# B&R Automation Studio project SysReset
Automation Studio 4.9

## Configuration TestSetup

CPU X20CP1585, AutomationRuntime C4.90, Build 4.1.2, Vc V4.72.0

### Task classes (Cpu.sw)
```
Cyclic#4:
  DevLinker <- DevLinker.prg
  SysRst <- SysRst.prg
Cyclic#7:
  HelloFile <- HelloFile.prg
Binaries: FWRules, TCData, udbdef, asfw, User, iomap, sysconf, arconfig, ashwd, Role, ashwac
Libraries: sys_lib, runtime, standard, AsSem, FileIO, AsIODiag, asieccon, astime
```

### Hardware
```
X20BM11 : X20BM11 v1.0.0.1  [X2X1 -> X20CP1585.IF6]
X20CP1585 : X20CP1585 v1.8.1.0
  Connector IF2:
    ActivateDevice = 1
    HostName = sysreset
  ConfigurationID = SysReset_Config1
  Simulation = 1
  EthernetHostName = sysreset
  ActivateDns = 1
  GetDnsFromDhcp = 2
X20DI9371 : X20DI9371 v1.1.0.0  [SS1 -> X20TB12.SS; SL -> X20BM11.SL1]
X20TB12 : X20TB12 v1.0.0.0
```

### IoMap.iom - X20CP1585/IoMap.iom
```iecst
VAR_CONFIG
	::SysRst:diVdc24Ok AT %IX."X20DI9371".DigitalInput01;
END_VAR
```

### PvMap.vvm - X20CP1585/PvMap.vvm
```iecst
VAR_CONFIG
	::SysRst:oSemIdent AT %Q.::HelloFile:iSemIdent; (*Insert your comment here...*)
	::SysRst:oFileSystemLocked AT %Q.::HelloFile:iFileSystemLocked; (*Insert your comment here...*)
END_VAR
```

## Logical view

Binary libraries used (declarations not repeated): operator, runtime, astime, AsIecCon, sys_lib, standard, AsSem, FileIO, AsIODiag

### Global.var - Global variables
```iecst
VAR CONSTANT
	FILE_DEVICE_LOCAL : STRING[80] := 'LOCAL';
END_VAR
```


### Program Logical/DevLinker (IEC) - Creates file devices

#### Variables.var
```iecst
VAR
	fbDevLink : DevLink; (*links file device*)
	fbDevUnlink : DevUnlink; (*unlinks file device*)
	fbDirCreate : DirCreate; (*creates directory*)
END_VAR
VAR CONSTANT
	FILE_DEVICE_TEMP : STRING[80] := '__TEMP__'; (*name of temporary file device*)
END_VAR
```

#### Main.st
```iecst
(*********************************************************************************
 * Copyright: B&R Industrial Automation GmbH
 * Author:    knausenbergl
 * Created:   April 12, 2021/1:55 PM

Link a file device on the CF user partition (ArEmb) or in the windows temp folder (ArSim), respectively.
Required for file handling.
 *********************************************************************************)

PROGRAM _INIT

	(* for ArSim, create folder structure under "C:/Temp" *)
	IF DiagCpuIsARsim() OR DiagCpuIsSimulated() THEN
		(* link file device in windows temp folder. this file device is only needed for creating subfolders. *)
		fbDevLink.enable := TRUE;
		fbDevLink.pDevice := ADR(FILE_DEVICE_TEMP);
		fbDevLink.pParam := ADR('/DEVICE=C:/Temp/');
		fbDevLink();

		(* create directory "SysReset" in windows temp folder *)
		fbDirCreate.enable := TRUE;
		fbDirCreate.pDevice := ADR(FILE_DEVICE_TEMP);
		fbDirCreate.pName := ADR('SysReset');
		fbDirCreate();

		(* unlink temporary file device, it is no longer needed *)
		fbDevUnlink.enable := TRUE;
		fbDevUnlink.handle := fbDevLink.handle;
		fbDevUnlink();
	END_IF

	(* link FILE_DEVICE_LOCAL, which is used for data storage by other tasks *)
	fbDevLink.enable := TRUE;
	fbDevLink.pDevice := ADR(FILE_DEVICE_LOCAL);
	IF DiagCpuIsARsim() OR DiagCpuIsSimulated() THEN
		fbDevLink.pParam := ADR('/DEVICE=C:/Temp/SysReset');
	ELSE
		fbDevLink.pParam := ADR('/DEVICE=F:/');
	END_IF
	fbDevLink();

END_PROGRAM

PROGRAM _CYCLIC
	(* Insert code here *)

END_PROGRAM

PROGRAM _EXIT

	fbDevUnlink.enable := TRUE;
	fbDevUnlink.handle := fbDevLink.handle;
	fbDevUnlink();

END_PROGRAM
```

### Program Logical/SysRst (IEC) - Controlled PLC shutdown

#### Main.st - Init, cyclic, exit code
```iecst
(*********************************************************************************
 * Copyright: B&R Industrial Automation GmbH
 * Author:    knausenbergl
 * Created:   January 18, 2021/11:20 AM

This task initiates a controlled shutdown of the PLC if either of the following conditions applies:
1. Drop in 24VDC supply, running on buffered 24VDC supply. (Only applies if buffered 24VDC is used.)
2. Shutdown command triggered, e.g. by visualization.

This task ensures file consistency in the case of a shutdown. This is done via the use of
semaphores. Any task accessing the file system must acquire a semaphore. The shutdown only
starts if the semaphore is no longer in use.
 *********************************************************************************)

PROGRAM _INIT

	(* create semaphore for detecting usage of file system *)
	fbSemCreate.enable		:= TRUE;
	fbSemCreate.maxCount	:= SEM_MAX_COUNT;
	fbSemCreate.initCount	:= fbSemCreate.maxCount;
	fbSemCreate();
	oSemIdent	:= fbSemCreate.ident;

	TOF_Vdc24Ok.PT	:= VDC24_OK_OFF_DELAY;

END_PROGRAM

PROGRAM _CYCLIC

	TOF_Vdc24Ok(IN := diVdc24Ok);			//off-delay for "24VDC OK" signal to filter short drops in 24VDC power supply
	F_TRIG_Vdc24Ok(CLK := TOF_Vdc24Ok.Q);	//falling edge of filtered "24VDC OK" signal

	(* check if file system is busy *)
	fbSemGetInfo.enable	:= TRUE;
	fbSemGetInfo.ident	:= fbSemCreate.ident;
	fbSemGetInfo();
	FileSystemBusy	:= (fbSemGetInfo.maxCount <> fbSemGetInfo.curCount);

	(* state machine *)
	CASE State OF
		(* initial state after boot *)
		STATE_INIT:
			State := STATE_IDLE;

		(* idle, waiting for event *)
		STATE_IDLE:
			IF (F_TRIG_Vdc24Ok.Q OR iCmdShutdown) THEN
				iCmdShutdown	:= FALSE;
				State := STATE_AWAIT_FILESYS;
			END_IF

		(* wait for file system to finish *)
		STATE_AWAIT_FILESYS:
			IF NOT FileSystemBusy THEN
				State := STATE_SHUTDOWN;
			END_IF

		(* shutdown *)
		STATE_SHUTDOWN:
			SYSreset(enable := TRUE, mode := 16#11);	//start shutdown in mode 0x11: WARMSTART (no restart, only shutdown, waits for "power off", in connection with UPS)

	END_CASE

	(* set outputs depending on current state *)
	CASE State OF
		STATE_AWAIT_FILESYS, STATE_SHUTDOWN:
			oFileSystemLocked := TRUE;
		ELSE
			oFileSystemLocked := FALSE;
	END_CASE

END_PROGRAM

PROGRAM _EXIT

	fbSemDelete.enable	:= TRUE;
	fbSemDelete.ident	:= fbSemCreate.ident;
	fbSemDelete();

END_PROGRAM
```

#### Types.typ - Local data types
```iecst
TYPE
	StateEnum :
		(
		STATE_INIT,
		STATE_IDLE,
		STATE_AWAIT_FILESYS,
		STATE_SHUTDOWN
		);
END_TYPE
```

#### Variables.var - Local variables
```iecst
VAR
	TOF_Vdc24Ok : TOF; (*off-delay for "24VDC OK" signal to filter short drops in 24VDC power supply*)
	F_TRIG_Vdc24Ok : F_TRIG; (*falling edge detection*)
END_VAR
VAR CONSTANT
	VDC24_OK_OFF_DELAY : TIME := T#50ms; (*off-delay for "24VDC OK" signal to filter short drops in 24VDC power supply*)
END_VAR
VAR
	fbSemCreate : SemCreate; (*creates a semaphore to block file system in case of shutdown*)
	fbSemDelete : SemDelete; (*deletes semaphore*)
END_VAR
VAR CONSTANT
	SEM_MAX_COUNT : USINT := 128; (*maximum number of times the semaphore can be acquired*)
END_VAR
VAR
	fbSemGetInfo : SemGetInfo; (*gets info about semaphore*)
	FileSystemBusy : BOOL; (*file system is busy*)
	State : StateEnum; (*actual state in state machine*)
END_VAR
```

#### LocalFunctions.fun
```iecst
{REDUND_ERROR} FUNCTION_BLOCK UaSYSReset (*OPC UA method wrapper for SYSReset*) (*$GROUP=User,$CAT=User,$GROUPICON=User.png,$CATICON=User.png*)
	VAR_INPUT
		Mode : USINT;
		Delay : TIME;
	END_VAR
	VAR
		State : USINT;
		State_1 : USINT;
		UaSrv_MethodOperate_0 : UaSrv_MethodOperate;
		FirstCycleInState : BOOL;
		TON_Delay : TON;
	END_VAR
END_FUNCTION_BLOCK
```

#### UaSYSReset.st
```iecst
(* OPC UA method wrapper for SYSReset *)
FUNCTION_BLOCK UaSYSReset

	(* set flag when entering new state *)
	FirstCycleInState	:= (State <> State_1);
	State_1	:= State;

	(* state-machine *)
	CASE State OF

		(* idle *)
		0, 255:
			State	:= 1;

		(* check if method is called *)
		1:
			IF FirstCycleInState THEN
				UaSrv_MethodOperate_0.Action := UaMoa_CheckIsCalled;
				UaSrv_MethodOperate_0(Execute := FALSE);
				UaSrv_MethodOperate_0.MethodName	:= 'SysReset';
				UaSrv_MethodOperate_0.Execute		:= TRUE;
			END_IF

			UaSrv_MethodOperate_0();
			IF UaSrv_MethodOperate_0.Done THEN
				IF UaSrv_MethodOperate_0.IsCalled THEN
					State	:= 2;
				ELSE
					State	:= 0;
				END_IF
			ELSIF UaSrv_MethodOperate_0.Error THEN
				State	:= 255;
			END_IF

		(* confirm method call *)
		2:
			IF FirstCycleInState THEN
				UaSrv_MethodOperate_0.Action := UaMoa_Finished;
				UaSrv_MethodOperate_0(Execute := FALSE);
				UaSrv_MethodOperate_0.Execute		:= TRUE;
			END_IF

			UaSrv_MethodOperate_0();
			IF UaSrv_MethodOperate_0.Done THEN
				State	:= 3;
			ELSIF UaSrv_MethodOperate_0.Error THEN
				State	:= 255;
			END_IF

		(* delay SYSreset *)
		3:
			IF FirstCycleInState THEN
				TON_Delay(IN := FALSE);
				TON_Delay.PT	:= Delay;
				TON_Delay.IN	:= TRUE;
			END_IF

			TON_Delay();
			IF TON_Delay.Q THEN
				State	:= 4;
			END_IF

		(* call SYSreset *)
		4:
			SYSreset(enable := TRUE, mode := Mode);
			State	:= 0;

	END_CASE

END_FUNCTION_BLOCK
```

- Methods.uam (not shown)

#### Interface.var - not listed in the package file held
```iecst
VAR
	diVdc24Ok : BOOL; (*digital input: 24VDC supply OK.
TRUE: 24VDC supply OK
FALSE: 24VDC supply interrupted, running on buffered 24VDC.

if you are using a 24VDC buffer module, such as 0PB0200.1, connect this digital input to the "Power Good" output of the buffer module. otherwise, do not connect this input.*)
	iCmdShutdown : BOOL; (*visu command: start shutdown

set this variable to TRUE to start the shutdown. variable is automatically reset by the application.*)
	oSemIdent : UDINT; (*semaphore ident*)
	oFileSystemLocked : BOOL; (*file system locked, file access no longer allowed*)
END_VAR
```

### Program Logical/HelloFile (IEC) - Example task with file handling

#### Main.st - Init, cyclic, exit code
```iecst
(*********************************************************************************
 * Copyright: B&R Industrial Automation GmbH
 * Author:    knausenbergl
 * Created:   April 12, 2021/1:55 PM

This task creates a file 'HelloWorld.txt' and writes to it. When writing, this task acquires
a semaphore, thereby blocking any shutdown in SysRst. The shutdown is delayed until all
writing operations are complete.
A writing command is issued by setting iCmdWrite to TRUE.
 *********************************************************************************)

PROGRAM _INIT

	FileDevice := FILE_DEVICE_LOCAL;
	FileName := 'HelloWorld.txt';
	WriteData := 'HelloWorld$n';

	(* create a file (in case it does not already exist) *)
	fbFileCreate.enable := TRUE;
	fbFileCreate.pDevice := ADR(FileDevice);
	fbFileCreate.pFile := ADR(FileName);
	fbFileCreate();

	(* close the file opened by FileCreate *)
	fbFileClose.enable := TRUE;
	fbFileClose.ident := fbFileCreate.ident;
	fbFileClose();

END_PROGRAM

PROGRAM _CYCLIC

	(* main state machine *)
	CASE State OF

		(* inital state after boot *)
		STATE_INIT:
			State := STATE_IDLE;

		(* idle, waiting for command *)
		STATE_IDLE, STATE_ERROR:
			IF iCmdWrite AND NOT iFileSystemLocked THEN
				iCmdWrite := FALSE;
				(* acquire semaphore before writing *)
				IF (SemAcquire(iSemIdent) = ERR_OK) THEN
					State := STATE_OPENING;
				ELSE
					State := STATE_ERROR;
				END_IF
			END_IF

		(* opening file *)
		STATE_OPENING:
			fbFileOpen.enable := TRUE;
			fbFileOpen.mode := fiWRITE_ONLY;
			fbFileOpen.pDevice := ADR(FileDevice);
			fbFileOpen.pFile := ADR(FileName);
			fbFileOpen();

			CASE fbFileOpen.status OF
				ERR_FUB_BUSY:
					// pass
				ERR_OK:
					State := STATE_WRITING;
				ELSE
					SemRelease(iSemIdent);
					State := STATE_ERROR;
			END_CASE

		(* writing to file *)
		STATE_WRITING:
			fbFileWrite.enable := TRUE;
			fbFileWrite.ident := fbFileOpen.ident;
			fbFileWrite.len := LEN(WriteData);
			fbFileWrite.offset := fbFileOpen.filelen;
			fbFileWrite.pSrc := ADR(WriteData);
			fbFileWrite();

			CASE fbFileWrite.status OF
				ERR_FUB_BUSY:
					// pass
				ERR_OK:
					State := STATE_CLOSING;
				ELSE
					State := STATE_CLOSING_ERROR;
			END_CASE

		(* closing file (also after error) *)
		STATE_CLOSING, STATE_CLOSING_ERROR:
			fbFileClose.enable := TRUE;
			fbFileClose.ident := fbFileOpen.ident;
			fbFileClose();

			CASE fbFileClose.status OF
				ERR_FUB_BUSY:
					// pass
				ERR_OK:
					SemRelease(iSemIdent);
					IF State = STATE_CLOSING THEN
						State := STATE_IDLE;
					ELSE
						State := STATE_ERROR;
					END_IF
				ELSE
					SemRelease(iSemIdent);
					State := STATE_ERROR;
			END_CASE

	END_CASE

END_PROGRAM

PROGRAM _EXIT

	fbFileClose.enable := TRUE;
	fbFileClose.ident := fbFileOpen.ident;
	fbFileClose();

END_PROGRAM
```

#### Types.typ - Local data types
```iecst
TYPE
	StateEnum :
		(
		STATE_INIT,
		STATE_IDLE,
		STATE_OPENING,
		STATE_WRITING,
		STATE_CLOSING_ERROR,
		STATE_CLOSING,
		STATE_ERROR
		);
END_TYPE
```

#### Variables.var - Local variables
```iecst
VAR
	fbFileClose : FileClose;
	fbFileWrite : FileWrite;
	fbFileOpen : FileOpen;
	fbFileCreate : FileCreate;
	State : StateEnum;
	FileName : STRING[80];
	FileDevice : STRING[80];
	WriteData : STRING[80];
END_VAR
```

#### Interface.var
```iecst
VAR
	iCmdWrite : BOOL; (*command: write to file*)
	iSemIdent : UDINT; (*semaphore ident*)
	iFileSystemLocked : BOOL; (*file system locked, file access no longer allowed*)
END_VAR
```

Listed in the project but not available here: Logical/Global.typ
